PROGRAM MAIN
VAR
END_VAR



// Bachelor:
PRG_ScaledInputs();
PRG_ControllerMode();
PRG_Filter();
PRG_Timer();

// 2. MODUS-VALG (Kun ett program får skrive til fU)
IF G_Mode.bManual THEN
    // Her kjører vi manual-programmet ditt med joystick
	PRG_Manual_PF_Gradient();
    //PRG_TestHome();
ELSIF G_Mode.bAuto THEN
    // Her kjører vi auto-rampen (0.05m til 0.45m)
	//PRG_AutoRamp_GradientFiltered();
	//RampfUTest();
	fU_Testing();
    
ELSE
    // SIKKERHET: Hvis ingen modus er valgt, stopp kranen helt
    G_OPC.fU := 0.0;
END_IF

PRG_Output();
// PID - NOT created
// FeedForward - not created

END_PROGRAM

(* stored: Version 1.1.0.1
   POU MAIN: Id {95bd3131-5c67-452d-927e-7536941f7837}, SpecialFunc None *)
